(* IEC 61131-3 sources: plc_programming/Ejercicios/project_files/build, 2 files *)

(* ---- plc.st ---- *)
TYPE
  LOGLEVEL : (CRITICAL, WARNING, INFO, DEBUG) := INFO;
END_TYPE

FUNCTION_BLOCK LOGGER
  VAR_INPUT
    TRIG : BOOL;
    MSG : STRING;
    LEVEL : LOGLEVEL := INFO;
  END_VAR
  VAR
    TRIG0 : BOOL;
  END_VAR

  IF TRIG AND NOT TRIG0 THEN
  {{
   LogMessage(GetFbVar(LEVEL),(char*)GetFbVar(MSG, .body),GetFbVar(MSG, .len));
  }}
  END_IF;
  TRIG0:=TRIG;
END_FUNCTION_BLOCK

PROGRAM rele
  VAR
    BTN_INICIO : BOOL;
    BTN_PARO : BOOL;
    M_MOTOR : BOOL;
    MOTOR : BOOL;
  END_VAR

  M_MOTOR := NOT(BTN_PARO) AND (BTN_INICIO OR M_MOTOR);
  MOTOR := M_MOTOR;
END_PROGRAM

CONFIGURATION Config0

  RESOURCE Res0 ON PLC
    TASK task0(INTERVAL := T#20ms,PRIORITY := 0);
    PROGRAM instance0 WITH task0 : rele;
  END_RESOURCE
END_CONFIGURATION

(* ---- generated_plc.st ---- *)
PROGRAM rele
  VAR
    BTN_INICIO : BOOL;
    BTN_PARO : BOOL;
    M_MOTOR : BOOL;
    MOTOR : BOOL;
  END_VAR

  M_MOTOR := NOT(BTN_PARO) AND (BTN_INICIO OR M_MOTOR);
  MOTOR := M_MOTOR;
END_PROGRAM

CONFIGURATION Config0

  RESOURCE Res0 ON PLC
    TASK task0(INTERVAL := T#20ms,PRIORITY := 0);
    PROGRAM instance0 WITH task0 : rele;
  END_RESOURCE
END_CONFIGURATION
